KUKA KRL data list: trig.dat

&ACCESS RVO
&REL 74
DEFDAT trig PUBLIC

GLOBAL STRUC ST_R_TRIG BOOL x, xOld, Q
GLOBAL STRUC ST_F_TRIG BOOL x, xOld, Q
GLOBAL STRUC ST_X_TRIG BOOL x, xOld, RQ, FQ

ENDDAT
